% RSLogix 500 project PRACTISE-10.RSS, saved by version 8.30.00.16 %
PROJECT "UNTITLED"    % processor: MicroLogix 1000 %

PROGRAM FILES
  LAD 2 "MAIN_PROG"  16 rungs
  LAD 3 "USER_FAULT"  1 rungs
  LAD 4 "HSC_INT"  1 rungs
  LAD 5 "STI_INT"  1 rungs
  LAD 6, 7, 8, 9, 10, 11, 12, 13, 14, 15, 16: only END

DATA FILES
  O0 OUTPUT  1 elements
  I1 INPUT  2 elements
  S2 STATUS  33 elements
  B3 BINARY  32 elements
  T4 TIMER  40 elements
  C5 COUNTER  32 elements
  R6 CONTROL  16 elements
  N7 INTEGER  105 elements

LADDER 2 "MAIN_PROG"
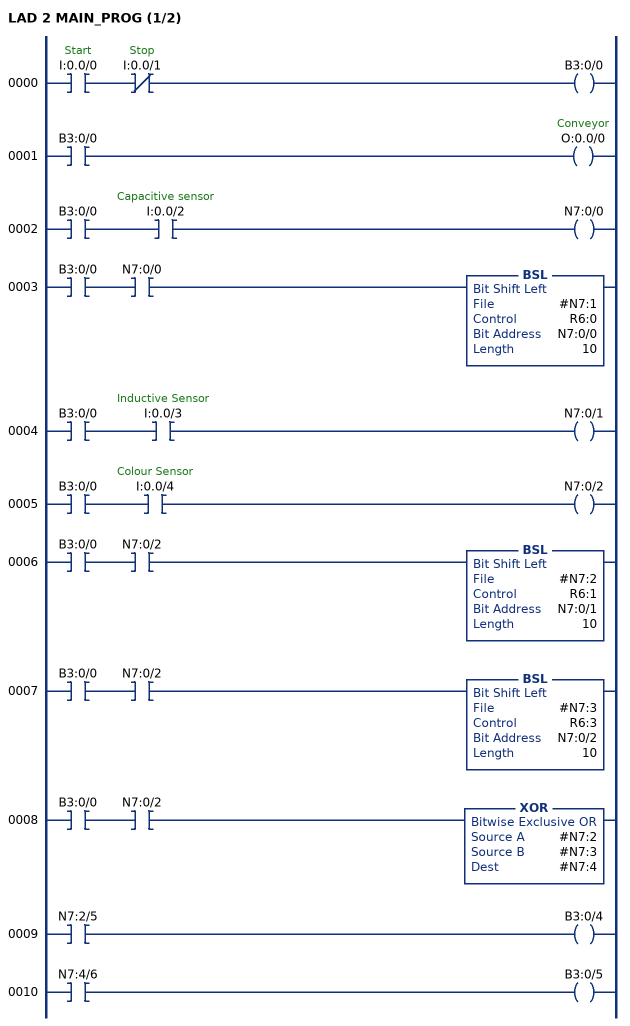
% Rung: 0 %
SOR XIC I:0.0/0 XIO I:0.0/1 OTE B3:0/0 EOR
%   I:0.0/0  "Start" %
%   I:0.0/1  "Stop" %
% Rung: 1 %
SOR XIC B3:0/0 OTE O:0.0/0 EOR
%   O:0.0/0  "Conveyor" %
% Rung: 2 %
SOR XIC B3:0/0 XIC I:0.0/2 OTE N7:0/0 EOR
%   I:0.0/2  "Capacitive sensor" %
% Rung: 3 %
SOR XIC B3:0/0 XIC N7:0/0 BSL #N7:1 R6:0 N7:0/0 10 EOR
% Rung: 4 %
SOR XIC B3:0/0 XIC I:0.0/3 OTE N7:0/1 EOR
%   I:0.0/3  "Inductive Sensor" %
% Rung: 5 %
SOR XIC B3:0/0 XIC I:0.0/4 OTE N7:0/2 EOR
%   I:0.0/4  "Colour Sensor" %
% Rung: 6 %
SOR XIC B3:0/0 XIC N7:0/2 BSL #N7:2 R6:1 N7:0/1 10 EOR
% Rung: 7 %
SOR XIC B3:0/0 XIC N7:0/2 BSL #N7:3 R6:3 N7:0/2 10 EOR
% Rung: 8 %
SOR XIC B3:0/0 XIC N7:0/2 XOR #N7:2 #N7:3 #N7:4 EOR
% Rung: 9 %
SOR XIC N7:2/5 OTE B3:0/4 EOR
% Rung: 10 %
SOR XIC N7:4/6 OTE B3:0/5 EOR

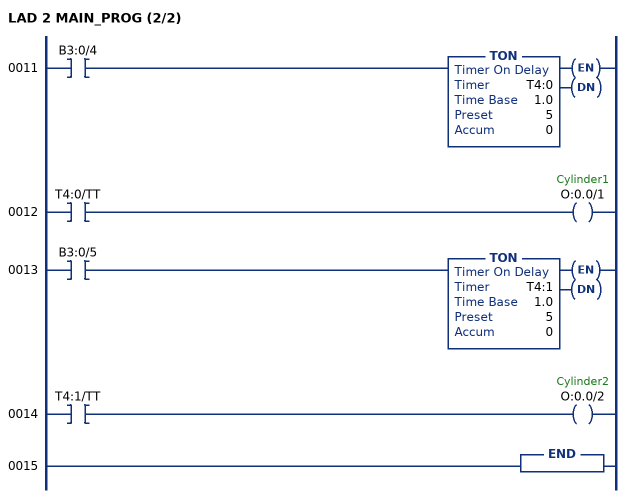
% Rung: 11 %
SOR XIC B3:0/4 TON T4:0 1.0 5 0 EOR
% Rung: 12 %
SOR XIC T4:0/TT OTE O:0.0/1 EOR
%   O:0.0/1  "Cylinder1" %
% Rung: 13 %
SOR XIC B3:0/5 TON T4:1 1.0 5 0 EOR
% Rung: 14 %
SOR XIC T4:1/TT OTE O:0.0/2 EOR
%   O:0.0/2  "Cylinder2" %
% Rung: 15 %
SOR END EOR

DATA TABLE (non-zero values as saved)
DATA T4
% .PRE .ACC %
% T4:0 % 5 0
% T4:1 % 5 0
% T4:3 % 5 0
DATA R6
% .LEN .POS %
% R6:0 % 10 0
% R6:1 % 10 0
% R6:2 % 10 0
% R6:3 % 10 0
